FUNCTION_BLOCK T_GripperProductionMode EXTENDS T_NamedBase IMPLEMENTS I_PackMode
VAR
	_gripper : I_GripperModule;
END_VAR

METHOD Initialise
VAR_INPUT
	Gripper : I_GripperModule;
END_VAR
_gripper := Gripper;
END_METHOD

END_FUNCTION_BLOCK

(* stored: Version 1.1.0.1, ProductVersion 3.1.4024.12
   POU T_GripperProductionMode: Id {512c3ca2-eafa-4ddf-99c9-0c6b8a984674}, SpecialFunc None
   Method Initialise: Id {0985137a-cccb-40be-b232-c3d89fe0c35b} *)
